// TIA Portal V16 export
// export: Created 2024-04-09T10:29:19.4917564Z, ExportSetting WithDefaults, DisplayName Totally Integrated Automation Portal, DisplayVersion V16 Update 3, DisplayName TIA Portal Version Control Interface, DisplayVersion V16 Update 2, DisplayName TIA Portal Openness, DisplayVersion V16 Update 3, DisplayName STEP 7 Professional, DisplayVersion V16 Update 3, DisplayName STEP 7 Safety, DisplayVersion V16, DisplayName WinCC Professional, DisplayVersion V16 Update 3
TYPE "UT00800_St_K_AnData"
TITLE = Static UDT [CONSTANTS] — Analog Card Ranges, Types and Coefficients
// PRACTICAL SERIES AUTOMATION LIBRARY (PAL)   —   COPYRIGHT 2020 – M. GLEDHILL (MIT LICENCE)
//                   ———— ◆ ————
// FULL ONLINE DOCUMENTATION IS AVAILABLE AT: https://practicalseries.com/2001-pal/index.html
// stored: IsFailsafeCompliant false
   STRUCT
      revInfo { ExternalWritable := 'False'} : "UT01000_St_SysRevision";   // ▀▀▀▀ UDT CURRENT REVISION
      ___________0010_0 { ExternalAccessible := 'False'; ExternalVisible := 'False'; ExternalWritable := 'False'} : Bool;
      ___________0010_1 { ExternalAccessible := 'False'; ExternalVisible := 'False'; ExternalWritable := 'False'} : Bool;   // ▀▀▀▀ AIO SIGNAL CODE
      AIO_CODE : UInt := 16#0000;   // Instrument code (type, coefficient and range)
      ___________0020_0 { ExternalAccessible := 'False'; ExternalVisible := 'False'; ExternalWritable := 'False'} : Bool := false;
      ___________0010_2 { ExternalAccessible := 'False'; ExternalVisible := 'False'; ExternalWritable := 'False'} : Bool;   // ▀▀▀▀ AIO RANGE DATA
      RAW_MIN : Int := 0;   // Minimum value of the analog input range
      RAW_MAX : Int := 27648;   // Maximum value of the analog input range
      RAW_NAME : String[60] := 'User defined instrument type';   // Signal type name
      ___________0030_1 { ExternalAccessible := 'False'; ExternalVisible := 'False'; ExternalWritable := 'False'} : Bool;
      ___________0030_2 { ExternalAccessible := 'False'; ExternalVisible := 'False'; ExternalWritable := 'False'} : Bool;   // ▀▀▀▀ AIO CARD PARAMETERS
      PARAM_TYPE : Byte := 16#00;   // Unique measurement type code
      PARAM_RANGE : Byte := 16#00;   // Unique measurement range code
      PARAM_COEF : Byte := 16#00;   // Unique temperature coefficient code (thermal resistance only)
      VALUE_COEF : Real;   // Temperature coefficient actual value, Ω/Ω/°C (thermal resistance only)
   END_STRUCT;
   // revInfo.REV_BLOCK := 'UT00800';
   // revInfo.REV_NUMBER := '000.101';
   // revInfo.REV_DATE := '2024-04-09';
   // revInfo.REV_AUTHOR := 'M. Gledhill';
END_TYPE
